INTERFACE IStation

METHOD FindMoverMatch : udint
VAR_INPUT
END_VAR
END_METHOD

METHOD FindNextPosition : IPosition;
VAR_INPUT
END_VAR
END_METHOD

METHOD GetMovers : BOOL
VAR_INPUT
END_VAR
END_METHOD

METHOD SetPosRef : BOOL
VAR_INPUT
	PosIndex : DINT;
	PosRef	: REFERENCE TO FB_PositionX;
END_VAR
END_METHOD

METHOD SetStationAttraction : BOOL
VAR_INPUT
	setState : INT;
END_VAR
END_METHOD

METHOD SetTrackRef : BOOL
VAR_INPUT
	TrackRef : ITrackList;
END_VAR
END_METHOD

END_INTERFACE

(* stored: Version 1.1.0.1, ProductVersion 3.1.4026.12
   Itf IStation: Id {ad2a9605-1431-4e38-b464-9e75dcc5c264}
   Method FindMoverMatch: Id {3d014b2b-d53b-460d-a169-a1d3bd4aeeed}
   Method FindNextPosition: Id {416cc32a-58cf-4c57-bedd-4ac90c640b8e}
   Method GetMovers: Id {5dcd5f5f-d1a7-4570-849e-96d9cadb4164}
   Method SetPosRef: Id {afdd7a2b-b162-4d22-a4b7-f5bf1a15001e}
   Method SetStationAttraction: Id {52188779-1db2-452f-ac2a-630123340e7a}
   Method SetTrackRef: Id {14a6e016-9a08-4024-88a3-d8555f33dd0f} *)
